# EPICS autosave request: stdApp/Db/scalerSoftCtrl_settings.req
file transform_settings.req P=$(P)$(Q)Tran
